PROGRAM MAIN_RCT
VAR
END_VAR


RULLI_CENTRO_TAGLI();

END_PROGRAM

(* stored: Version 1.1.0.1, ProductVersion 3.1.4022.12
   POU MAIN_RCT: Id {9137ec8f-ca65-46e8-8263-25de0e63dc7a}, SpecialFunc None *)
